FUNCTION F_IsOverheat : BOOL
VAR_INPUT
	 rTemp : REAL; 
END_VAR
VAR
END_VAR


F_IsOverheat := rTemp > 80.0;

END_FUNCTION

(* stored: Version 1.1.0.1, ProductVersion 3.1.4024.16
   POU F_IsOverheat: Id {77c2eefc-c493-4b8f-9922-a172f92317d1}, SpecialFunc None *)
